FUNCTION_BLOCK FB_Drum IMPLEMENTS  ITF_Device
VAR_INPUT
END_VAR
VAR_OUTPUT
END_VAR
VAR
	_stCBMLInfo 	: stCBMLInfo;
END_VAR

{warning 'add method implementation '}
METHOD M_GetState : BOOL;

VAR_OUTPUT
	O_stCBMLInfo : stCBMLInfo;
END_VAR
O_stCBMLInfo := _stCBMLInfo;
END_METHOD

{warning 'add method implementation '}
METHOD M_SetName : BOOL
VAR_INPUT
	sName	: STRING;
END_VAR
_stCBMLInfo.sName := sName;
END_METHOD

{warning 'add property implementation'}
PROPERTY P_stCBMLInfo : stCBMLInfo
GET
P_stCBMLInfo := _stCBMLInfo;
END_GET
SET
END_SET
END_PROPERTY

END_FUNCTION_BLOCK

(* stored: Version 1.1.0.1, ProductVersion 3.1.4024.11
   POU FB_Drum: Id {7fac3d5d-3198-46cf-8f5c-d234e1b9f4fb}, SpecialFunc None
   Method M_GetState: Id {0b47d5c4-b465-4374-b22a-4dec1a011bcb}
   Method M_SetName: Id {590fa758-ff6e-49d8-a0d2-61a6a067b50a}
   Property P_stCBMLInfo: Id {70eea36c-bedd-4e8a-b706-270a8746cbd7}
   Get Get: Id {268b79f4-1a21-46a2-b126-fb0b59139a1e}
   Set Set: Id {8c3e1ada-5edb-4e03-a91a-1fe373d031b3} *)
